SYSTEM TANK_MVL (* Level Control System Model+View+HMI *)
  (* Standard: 61499-1; Classification: Simulation; ApplicationDomain: Process Control *)
  (* Version 0.0, 2004-09-01, JHC, Rockwell Automation, Extended from TANK_VIEWL *)
  DEVICE HMI : FRAME_DEVICE
    RESOURCE VALVE : PANEL_RESOURCE
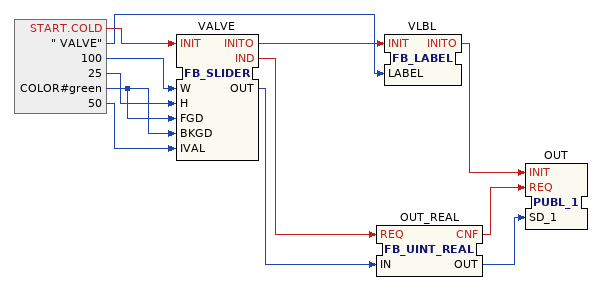
      FBS
        OUT : PUBL_1;
        VALVE : FB_SLIDER;
        VLBL : FB_LABEL;
        OUT_REAL : FB_UINT_REAL;
      END_FBS
      EVENT_CONNECTIONS
        START.COLD TO VALVE.INIT;
        VALVE.INITO TO VLBL.INIT;
        VLBL.INITO TO OUT.INIT;
        VALVE.IND TO OUT_REAL.REQ;
        OUT_REAL.CNF TO OUT.REQ;
      END_CONNECTIONS
      DATA_CONNECTIONS
        " VALVE" TO VLBL.LABEL;
        100 TO VALVE.W;
        25 TO VALVE.H;
        COLOR#green TO VALVE.FGD;
        VALVE.OUT TO OUT_REAL.IN;
        OUT_REAL.OUT TO OUT.SD_1;
        COLOR#green TO VALVE.BKGD;
        50 TO VALVE.IVAL;
      END_CONNECTIONS
    END_RESOURCE
    RESOURCE PUMP : PANEL_RESOURCE
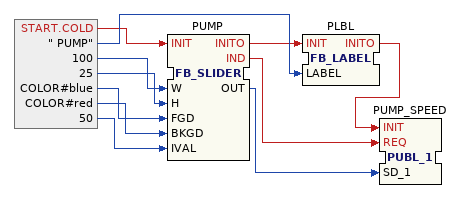
      FBS
        PUMP_SPEED : PUBL_1;
        PUMP : FB_SLIDER;
        PLBL : FB_LABEL;
      END_FBS
      EVENT_CONNECTIONS
        PUMP.INITO TO PLBL.INIT;
        PLBL.INITO TO PUMP_SPEED.INIT;
        START.COLD TO PUMP.INIT;
        PUMP.IND TO PUMP_SPEED.REQ;
      END_CONNECTIONS
      DATA_CONNECTIONS
        " PUMP" TO PLBL.LABEL;
        100 TO PUMP.W;
        25 TO PUMP.H;
        PUMP.OUT TO PUMP_SPEED.SD_1;
        COLOR#blue TO PUMP.FGD;
        COLOR#red TO PUMP.BKGD;
        50 TO PUMP.IVAL;
      END_CONNECTIONS
    END_RESOURCE
  END_DEVICE
  DEVICE RECORDER : FRAME_DEVICE
    RESOURCE RES1 : PANEL_RESOURCE
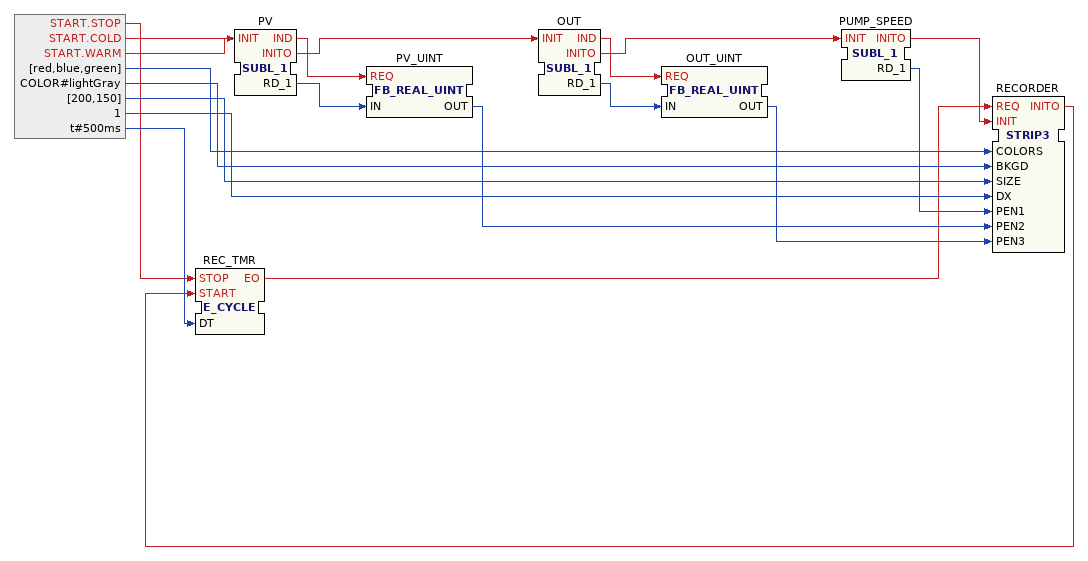
      FBS
        PUMP_SPEED : SUBL_1;
        PV : SUBL_1;
        OUT : SUBL_1;
        RECORDER : STRIP3;
        REC_TMR : E_CYCLE;
        PV_UINT : FB_REAL_UINT;
        OUT_UINT : FB_REAL_UINT;
      END_FBS
      EVENT_CONNECTIONS
        START.STOP TO REC_TMR.STOP;
        REC_TMR.EO TO RECORDER.REQ;
        PV.IND TO PV_UINT.REQ;
        OUT.IND TO OUT_UINT.REQ;
        START.COLD TO PV.INIT;
        START.WARM TO PV.INIT;
        PV.INITO TO OUT.INIT;
        OUT.INITO TO PUMP_SPEED.INIT;
        PUMP_SPEED.INITO TO RECORDER.INIT;
        RECORDER.INITO TO REC_TMR.START;
      END_CONNECTIONS
      DATA_CONNECTIONS
        [red,blue,green] TO RECORDER.COLORS;
        COLOR#lightGray TO RECORDER.BKGD;
        [200,150] TO RECORDER.SIZE;
        1 TO RECORDER.DX;
        t#500ms TO REC_TMR.DT;
        PUMP_SPEED.RD_1 TO RECORDER.PEN1;
        PV.RD_1 TO PV_UINT.IN;
        PV_UINT.OUT TO RECORDER.PEN2;
        OUT.RD_1 TO OUT_UINT.IN;
        OUT_UINT.OUT TO RECORDER.PEN3;
      END_CONNECTIONS
    END_RESOURCE
  END_DEVICE
  DEVICE MV : FRAME_DEVICE (* Model+View *)
    RESOURCE TANK_MDL : EMB_RES
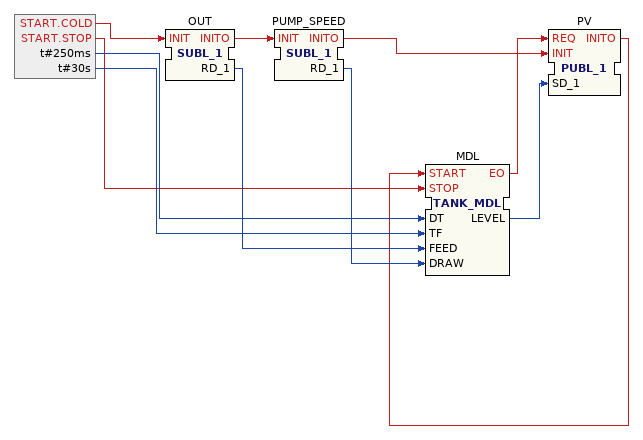
      FBS
        MDL : TANK_MDL;
        PUMP_SPEED : SUBL_1;
        OUT : SUBL_1;
        PV : PUBL_1;
      END_FBS
      EVENT_CONNECTIONS
        START.COLD TO OUT.INIT;
        OUT.INITO TO PUMP_SPEED.INIT;
        MDL.EO TO PV.REQ;
        START.STOP TO MDL.STOP;
        PUMP_SPEED.INITO TO PV.INIT;
        PV.INITO TO MDL.START;
      END_CONNECTIONS
      DATA_CONNECTIONS
        PUMP_SPEED.RD_1 TO MDL.DRAW;
        t#250ms TO MDL.DT;
        OUT.RD_1 TO MDL.FEED;
        t#30s TO MDL.TF;
        MDL.LEVEL TO PV.SD_1;
      END_CONNECTIONS
    END_RESOURCE
    RESOURCE PUMP_MDL : EMB_RES
      FBS
        MDL : SHAFT_MDL;
        PUMP_POS : PUBL_1;
        PUMP_SPEED : SUBL_1;
        UNSC : UNSCALE;
      END_FBS
      EVENT_CONNECTIONS
        START.COLD TO PUMP_SPEED.INIT;
        PUMP_SPEED.INITO TO PUMP_POS.INIT;
        MDL.EO TO PUMP_POS.REQ;
        PUMP_POS.INITO TO MDL.START;
        PUMP_SPEED.IND TO UNSC.REQ;
      END_CONNECTIONS
      DATA_CONNECTIONS
        t#100ms TO MDL.DT;
        MDL.POS TO PUMP_POS.SD_1;
        UNSC.OUT TO MDL.V;
        PUMP_SPEED.RD_1 TO UNSC.IN;
        360 TO UNSC.MAX;
      END_CONNECTIONS
    END_RESOURCE
    RESOURCE VALVE : VIEW_PANEL
      FBS
        OUT : SUBL_1;
        VALVE : VALVE_VIEW;
        OUT_UINT : FB_REAL_UINT;
      END_FBS
      EVENT_CONNECTIONS
        START.COLD TO OUT.INIT;
        OUT.INITO TO VALVE.INIT;
        OUT.IND TO OUT_UINT.REQ;
        OUT_UINT.CNF TO VALVE.REQ;
      END_CONNECTIONS
      DATA_CONNECTIONS
        50 TO VALVE.DIA;
        [0,255,0] TO VALVE.FGD;
        OUT.RD_1 TO OUT_UINT.IN;
        OUT_UINT.OUT TO VALVE.POS;
      END_CONNECTIONS
    END_RESOURCE
    RESOURCE TANK : VIEW_PANEL
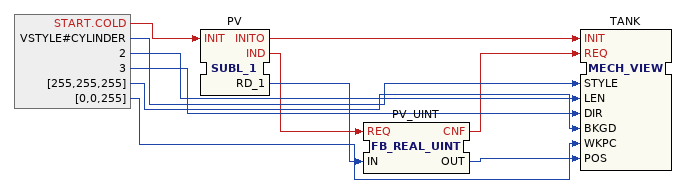
      FBS
        TANK : MECH_VIEW;
        PV : SUBL_1;
        PV_UINT : FB_REAL_UINT;
      END_FBS
      EVENT_CONNECTIONS
        PV.INITO TO TANK.INIT;
        START.COLD TO PV.INIT;
        PV.IND TO PV_UINT.REQ;
        PV_UINT.CNF TO TANK.REQ;
      END_CONNECTIONS
      DATA_CONNECTIONS
        VSTYLE#CYLINDER TO TANK.STYLE;
        2 TO TANK.LEN;
        3 TO TANK.DIR;
        [255,255,255] TO TANK.BKGD;
        [0,0,255] TO TANK.WKPC;
        PV.RD_1 TO PV_UINT.IN;
        PV_UINT.OUT TO TANK.POS;
      END_CONNECTIONS
    END_RESOURCE
    RESOURCE PUMP : VIEW_PANEL
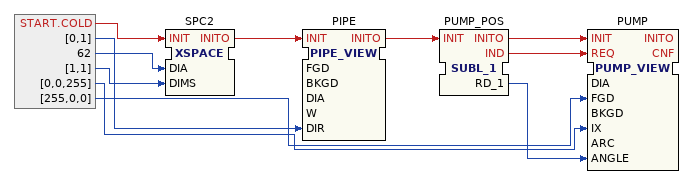
      FBS
        PUMP_POS : SUBL_1;
        SPC2 : XSPACE;
        PIPE : PIPE_VIEW;
        PUMP : PUMP_VIEW;
      END_FBS
      EVENT_CONNECTIONS
        SPC2.INITO TO PIPE.INIT;
        START.COLD TO SPC2.INIT;
        PIPE.INITO TO PUMP_POS.INIT;
        PUMP_POS.INITO TO PUMP.INIT;
        PUMP_POS.IND TO PUMP.REQ;
      END_CONNECTIONS
      DATA_CONNECTIONS
        [0,1] TO PIPE.DIR;
        62 TO SPC2.DIA;
        [1,1] TO SPC2.DIMS;
        PUMP_POS.RD_1 TO PUMP.ANGLE;
        [0,0,255] TO PUMP.IX;
        [255,0,0] TO PUMP.FGD;
      END_CONNECTIONS
    END_RESOURCE
    DATA_CONNECTIONS
      [1,2] TO TANK.SIZE;
      75 TO TANK.DIA;
      50 TO PUMP.DIA;
      [4,1] TO PUMP.SIZE;
      50 TO VALVE.DIA;
      [1,3] TO VALVE.SIZE;
    END_CONNECTIONS
  END_DEVICE
  DATA_CONNECTIONS (* parameter values *)
    [100,100,210,100] TO HMI.BOUNDS;
    [2,1] TO HMI.GRID;
    [310,100,175,250] TO MV.BOUNDS;
    [100,200,210,200] TO RECORDER.BOUNDS;
  END_CONNECTIONS
END_SYSTEM
